FUNCTION_BLOCK FB_MovingAverageInt
VAR_INPUT
	ValueToAdd : UINT;
END_VAR
VAR_IN_OUT
	AverageArray  : ARRAY [*] OF UINT;
END_VAR
VAR_OUTPUT
	CurrentValue : UINT;
END_VAR
VAR
	CurrentIndex : UINT;
	NumValues : UINT;
END_VAR
VAR_TEMP
	I: DINT;
	Sum: UDINT;
	ArrayLength : UINT;
END_VAR

// Compute average over array.
// The order of this addition and MOD are important to avoid going out of bounds.
ArrayLength := TO_UINT(UPPER_BOUND(AverageArray, 1) - LOWER_BOUND(AverageArray, 1) + 1);
AverageArray[CurrentIndex] := ValueToAdd;
CurrentIndex := CurrentIndex + 1;
CurrentIndex := CurrentIndex MOD ArrayLength;
NumValues := MIN(NumValues + 1 , ArrayLength);
// This wastes a little time walking pointless values if the array is underfilled,
// but they are zero initialized and thus should not afffect the calculation.
FOR I := LOWER_BOUND(AverageArray, 1) TO UPPER_BOUND(AverageArray, 1) BY 1 DO
	Sum := Sum + AverageArray[I];
END_FOR
CurrentValue := TO_UINT(Sum / NumValues);

END_FUNCTION_BLOCK

(* stored: Version 1.1.0.1, ProductVersion 3.1.4022.16
   POU FB_MovingAverageInt: Id {85bab29d-2c07-4c5a-a127-c5ff6504e896}, SpecialFunc None *)
